// TIA Portal V21 program export: 1 tag tables, 0 data types, 0 data blocks, 2 code blocks (in call order from the OBs), 0 instance data blocks

VAR_GLOBAL   // PLC tag table "Default tag table"
   Start AT %I0.0 : Bool;   // Start Button
   AutoON AT %I0.1 : Bool;   // Process Running
   Stop AT %I0.2 : Bool;   // Stop Button
   EmgStop AT %I0.3 : Bool;   // Emergency Stop
   Valve AT %Q1.0 : Bool;   // Control Valve
END_VAR

ORGANIZATION_BLOCK "Main"   // OB1, LAD, ProgramCycle
TITLE = "Main Program Sweep (Cycle)"
{ S7_Optimized_Access := 'TRUE' }
// stored: SetENOAutomatically false
   VAR_INPUT
      Initial_Call : Bool;   // Initial call of this OB
      Remanence : Bool;   // =True, if remanent data are available
   END_VAR
BEGIN

REGION Network 1: Safety
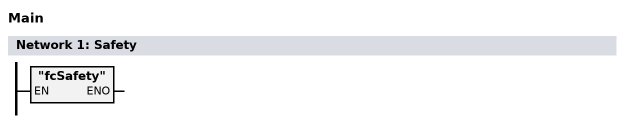
   RUNG wire#powerrail
      "fcSafety"()
   END_RUNG
   // the same network as SCL:
   "fcSafety"();
END_REGION
END_ORGANIZATION_BLOCK

FUNCTION "fcSafety" : Void   // FC1, LAD
{ S7_Optimized_Access := 'TRUE' }
// stored: SetENOAutomatically false
BEGIN

REGION Network 1: Safety
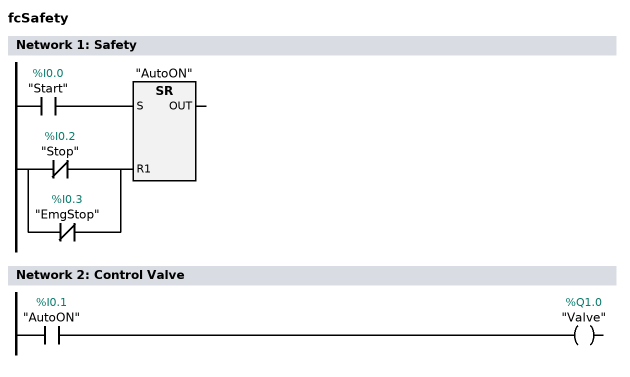
   RUNG wire#powerrail
      Contact( "Start" )
      S_SR(operand := "AutoON", r1 := wire#w1)
   END_RUNG
   RUNG wire#powerrail
      I_Contact( "Stop" )
   END_RUNG wire#w1
   RUNG wire#powerrail
      I_Contact( "EmgStop" )
   END_RUNG wire#w1
   // the same network as SCL:
   IF "Start" THEN
       "AutoON" := TRUE;   // SR flip-flop
   END_IF;
   IF NOT "Stop" OR NOT "EmgStop" THEN "AutoON" := FALSE; END_IF;
END_REGION

REGION Network 2: Control Valve
   RUNG wire#powerrail
      Contact( "AutoON" )
      Coil( "Valve" )
   END_RUNG
   // the same network as SCL:
   "Valve" := "AutoON";
END_REGION
END_FUNCTION
